{attribute 'GeneratedUsingTerminal: EM7004-0000-9996'}
{attribute addProperty BoxType "EM7004-0000-9996"}
{attribute addProperty Id "Enable_PLSAT %Q*BOOL1"}
{attribute addProperty CRC "2948061941"}
{attribute addProperty Size "1"}
TYPE PLS_Outputs_AFB7DAF5 :
STRUCT
	{attribute addProperty Name "Enable_PLS"}
	Enable_PLS AT %Q* : BOOL;
END_STRUCT
END_TYPE

(* stored: Version 1.2.0.0, ProductVersion 3.1.4024.9
   DUT PLS_Outputs_AFB7DAF5: Id {0d33ff66-c744-48aa-8db1-8581c9fdd9e4} *)
